% RSLogix 500 project P1_MARTIN_I.RSS, saved by version 8.30.00.16 %
PROJECT "UNTITLED"    % processor: Bul.1763 MicroLogix 1100 Series B %

PROGRAM FILES
  LAD 2 "MAIN"  3 rungs
  LAD 3 "DIGITAL IO"  5 rungs
  LAD 5 "CONTROLS"  6 rungs

DATA FILES
  O0 OUTPUT  5 elements
  I1 INPUT  7 elements
  S2 STATUS  66 elements
  B3 BINARY  1 elements
  T4 TIMER  1 elements
  C5 COUNTER  1 elements
  R6 CONTROL  1 elements
  N7 INTEGER  2 elements
  F8 FLOAT  1 elements

LADDER 2 "MAIN"
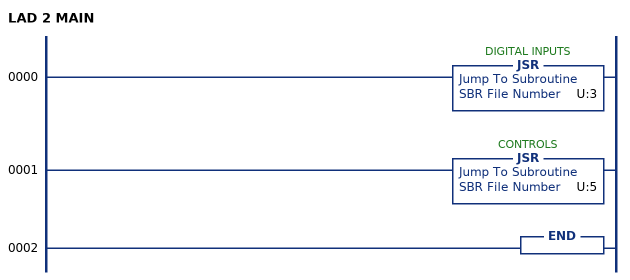
% Rung: 0 %
SOR JSR U:3 EOR
%   U:3  "DIGITAL INPUTS" %
% Rung: 1 %
SOR JSR U:5 EOR
%   U:5  "CONTROLS" %
% Rung: 2 %
SOR END EOR

LADDER 3 "DIGITAL IO"
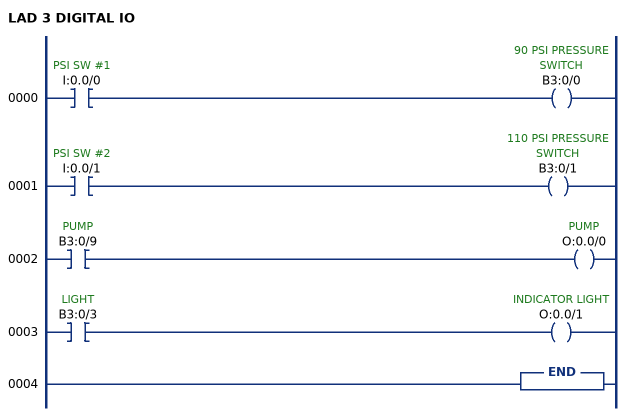
% Rung: 0 %
SOR XIC I:0.0/0 OTE B3:0/0 EOR
%   I:0.0/0  "PSI SW #1" %
%   B3:0/0  "90 PSI PRESSURE SWITCH" %
% Rung: 1 %
SOR XIC I:0.0/1 OTE B3:0/1 EOR
%   I:0.0/1  "PSI SW #2" %
%   B3:0/1  "110 PSI PRESSURE SWITCH" %
% Rung: 2 %
SOR XIC B3:0/9 OTE O:0.0/0 EOR
%   B3:0/9  "PUMP" %
%   O:0.0/0  "PUMP" %
% Rung: 3 %
SOR XIC B3:0/3 OTE O:0.0/1 EOR
%   B3:0/3  "LIGHT" %
%   O:0.0/1  "INDICATOR LIGHT" %
% Rung: 4 %
SOR END EOR

LADDER 5 "CONTROLS"
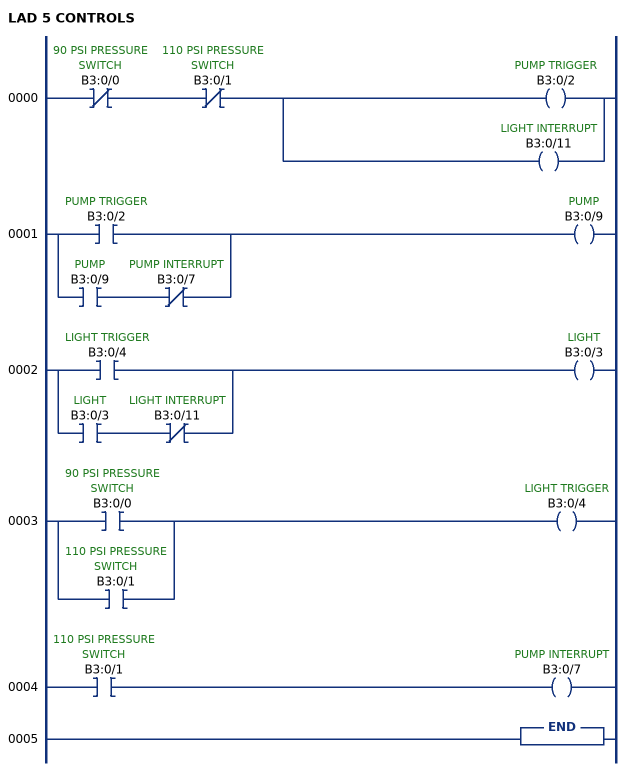
% Rung: 0 %
SOR XIO B3:0/0 XIO B3:0/1 BST OTE B3:0/2 NXB OTE B3:0/11 BND EOR
%   B3:0/0  "90 PSI PRESSURE SWITCH" %
%   B3:0/1  "110 PSI PRESSURE SWITCH" %
%   B3:0/2  "PUMP TRIGGER" %
%   B3:0/11  "LIGHT INTERRUPT" %
% Rung: 1 %
SOR BST XIC B3:0/2 NXB XIC B3:0/9 XIO B3:0/7 BND OTE B3:0/9 EOR
%   B3:0/2  "PUMP TRIGGER" %
%   B3:0/9  "PUMP" %
%   B3:0/7  "PUMP INTERRUPT" %
% Rung: 2 %
SOR BST XIC B3:0/4 NXB XIC B3:0/3 XIO B3:0/11 BND OTE B3:0/3 EOR
%   B3:0/4  "LIGHT TRIGGER" %
%   B3:0/3  "LIGHT" %
%   B3:0/11  "LIGHT INTERRUPT" %
% Rung: 3 %
SOR BST XIC B3:0/0 NXB XIC B3:0/1 BND OTE B3:0/4 EOR
%   B3:0/0  "90 PSI PRESSURE SWITCH" %
%   B3:0/1  "110 PSI PRESSURE SWITCH" %
%   B3:0/4  "LIGHT TRIGGER" %
% Rung: 4 %
SOR XIC B3:0/1 OTE B3:0/7 EOR
%   B3:0/1  "110 PSI PRESSURE SWITCH" %
%   B3:0/7  "PUMP INTERRUPT" %
% Rung: 5 %
SOR END EOR

OTHER DOCUMENTED ADDRESSES
  B3:0/5  "SYSTEM ENERGIZED"
  B3:0/6  "PUMP DE-ENERGIZE"
  B3:0/10  "ONE SHOT"
  B3:0/12  "ONE SHOT"
  I:0.0  "PSI SW #1"
  N7:0  "90 PSI SWITCH"
  N7:0/0  "90 PSI SWITCH"
  N7:0/1  "110 PSI PRESSURE SWITCH"
  N7:1  "110 PSI PRESSURE SWITCH"
  U:4  "DIGITAL OUTPUTS"
  U:6  "ALARMS"
